// TwinCAT 3 PLC project Untitled1
// ProgramVersion: 3.1.4024.0
// libraries:
//   Tc2_EtherCAT, * (Beckhoff Automation GmbH)
//   Tc2_IoFunctions, * (Beckhoff Automation GmbH)
//   Tc2_Standard, * (Beckhoff Automation GmbH)
//   Tc2_System, * (Beckhoff Automation GmbH)
//   Tc2_Utilities, * (Beckhoff Automation GmbH)
//   Tc3_EventLogger, * (Beckhoff Automation GmbH)
//   Tc3_Module, * (Beckhoff Automation GmbH)
// project tree:
//   / GlobalTextList.TcGTLO, PlcTask.TcTTO, Visualization Manager.TcVMO (not stored), VISU_TASK.TcTTO
//   GVLs/ GVL.TcGVL
//   POUs/EL6910/ FB_SafeDiag_Diagnostic.TcPOU, PH_SafeDiag_DiagHistory_black.TcVIS, PH_SafeDiag_Diagnostic_black.TcVIS, P_Sample.TcPOU, V_SafeDiag_Main.TcVIS
//   POUs/EL6910/Internal/Dedicated/DUTs/ E_SafeLogicState.TcTLEO, ST_EL6910_SafeDiag.TcDUT, ST_SafeDiag_HardwareInfos.TcDUT, ST_SafeDiag_SafetyProjectInfos.TcDUT, ST_SafeDiag_VisualisationInfos.TcDUT
//   POUs/EL6910/Internal/Dedicated/FBs/ FB_HardwareInfos.TcPOU, FB_SafeDiag_Visualisation.TcPOU, FB_SafetyProjectInfos.TcPOU
//   POUs/EL6910/Internal/General/DiagHistory_Events/ FB_DiagHistory_Listener.TcPOU, GVL_DiagHistory_SafetyEvents.TcGVL, ST_DiagHistory_Event.TcDUT
//   POUs/EL6910/Internal/General/EtherCAT/ FB_ReadSlaveBasicInformations.TcPOU, ST_EtherCat_SlaveBasicInfos.TcDUT
//   POUs/EL6910/Internal/General/SafetyEvents/ FB_Listener.TcPOU, FB_SafetyEvents.TcPOU, GVL_SafetyEvents.TcGVL, ST_Event.TcDUT
//   POUs/ MAIN.TcPOU
// real-time tasks:
//   TASK PlcTask: cycle T#10ms, priority 20, ADS port 350
//   TASK VISU_TASK: cycle T#200000us, priority 30, ADS port 351
// I/O:
//   DEVICE Device 1 (EtherCAT), AmsNetId 5.36.73.62.2.1
//     Term 1 (EK1200) [EK1200-5000 EtherCAT Power supply (2A E-Bus)]
//       Term 2 (EL1008) [EL1008 8Ch. Dig. Input 24V, 3ms]
//       Term 3 (EL2008) [EL2008 8Ch. Dig. Output 24V, 0.5A]
//       Term 4 (EL5151) [EL5151 1Ch. Inc. Encoder]
//       Term 5 (EL9110) [EL9110 Power Supplier with LED (24V, Diagnostics)]
//       Term 6 (EL6910) [EL6910, TwinSAFE PLC]
//       Term 7 (EL7037) [EL7037 1Ch. Stepper motor output stage (24V, 1.5A)]
//       Term 8 (EL9512) [EL9512 Power supply terminal 12V]
//       Term 9 (EL3162) [EL3162 2Ch. Ana. Input 0-10V]
//       Term 10 (EL4102) [EL4102 2Ch. Ana. Output  0-10V, 16bit]
//       Term 11 (EK1122) [EK1122 2 port EtherCAT junction]
//         Term 12 (EK1100) [EK1100 EtherCAT Coupler (2A E-Bus)]
//           Term 13 (EL1859) [EL1859 8Ch. Dig. Input 24V, 3ms, 8Ch. Dig. Output 24V, 0.5A]
//           Term 14 (EL1904) [EL1904, 4 Ch. Safety Input 24V, TwinSAFE]
//             modules: Module 1 (FSOES)
//           Term 15 (EL2904) [EL2904, 4 Ch. Safety Output 24V, 0.5A, TwinSAFE]
//             modules: Module 1 (FSOES), Module 2 (DO)
//           Term 16 (EL9110) [EL9110 Power Supplier with LED (24V, Diagnostics)]
//           Term 17 (EL2004) [EL2004 4Ch. Dig. Output 24V, 0.5A]
//           Term 18 (EL9410) [EL9410 E-Bus Power Supplier  (Diagnostics)]
//           Term 19 (EL7201-0010) [EL7201-0010 1Ch. MDP742 Servo motor output stage with OCT (50V, 4A)]
//           Term 27 (EL9011) [EL9011 End Terminal]
//         Term 20 (EK1101) [EK1101 EtherCAT Coupler (2A E-Bus, ID switch)]
//           Term 21 (EL1904) [EL1904, 4 Ch. Safety Input 24V, TwinSAFE]
//             modules: Module 1 (FSOES)
//           Term 22 (EL1252) [EL1252 2Ch. Fast Dig. Input 24V, 1µs, DC Latch]
//           Term 23 (EL1262) [EL1262 2Ch. Dig. Input 24V, 1µs, DC Oversample]
//           Term 24 (EL2252) [EL2252 2Ch. Dig. Output 24V, 0.5A, DC Time Stamp]
//           Term 25 (EL3702) [EL3702 2Ch. Ana. Input +/-10V, DIFF, Oversample]
//           Term 26 (EL4732) [EL4732 2Ch. Ana. Output +/-10V, Oversample]
//           Term 28 (EL9011) [EL9011 End Terminal]
// variable links:
//   Device 1 (EtherCAT) <-> Device 1 (EtherCAT)/Term 1 (EK1200)/Term 11 (EK1122)/Term 12 (EK1100)/Term 15 (EL2904)
//     Term 1 (EK1200)/Term 6 (EL6910)/ConnectionInputs/TwinSafeGroup1.Term 9 (EL2904) - Module 1 (FSOES)_3 TxPDO <-> Module 1 (FSOES)/RxPDO/FSOE
//   Device 1 (EtherCAT) <-> Device 1 (EtherCAT)/Term 1 (EK1200)/Term 6 (EL6910)
//     Term 1 (EK1200)/Term 11 (EK1122)/Term 12 (EK1100)/Term 15 (EL2904)/Module 1 (FSOES)/TxPDO/FSOE <-> ConnectionOutputs/TwinSafeGroup1.Term 9 (EL2904) - Module 1 (FSOES)_3 RxPDO
//   Untitled1/Untitled1 Instance <-> Device 1 (EtherCAT)/Term 1 (EK1200)/Term 6 (EL6910)
//     PlcTask Outputs/GVL.bErrAck <-> StandardOutputs/TwinSafeGroup1.ErrorAcknowledgement_1
//     PlcTask Outputs/GVL.bRun <-> StandardOutputs/TwinSafeGroup1.Run_2

CONFIGURATION Untitled1
    RESOURCE PLC ON TwinCAT3
        TASK PlcTask(INTERVAL := T#10ms, PRIORITY := 20);
        TASK VISU_TASK(INTERVAL := T#200000us, PRIORITY := 30);
        PROGRAM MAIN WITH PlcTask : MAIN;
        PROGRAM VisuElems_Visu_Prg WITH VISU_TASK : VisuElems.Visu_Prg;
    END_RESOURCE
END_CONFIGURATION

// ---- POUs/EL6910/Internal/Dedicated/DUTs/E_SafeLogicState.TcTLEO
{attribute 'qualified_only'}
{attribute 'strict'}
{attribute 'to_string'}
TYPE E_SafeLogicState :
(
	OFFLINE 		:= 0,
	RUN				:= 1,
	STOP			:= 2,
	SAFE			:= 3,
	ERROR           := 4,
	START           := 6,
	PREPARE         := 8,
	RESTORE         := 10,
	PROJECT_CRC_OK  := 11
);
END_TYPE

// ---- POUs/EL6910/Internal/Dedicated/DUTs/ST_EL6910_SafeDiag.TcDUT
TYPE ST_EL6910_SafeDiag :
STRUCT
	stBasicInfo						: ST_EtherCat_SlaveBasicInfos;									// EtherCAT slave basic infos
	stHardwareInfo					: ST_SafeDiag_HardwareInfos;									// Internal module hardware infos
	arrDiagHistory					: ARRAY [1.. GVL_SafetyEvents.MAX_EVENTS] OF ST_Event;			// Event Logger Listener
	stSafetyInfo					: ST_SafeDiag_SafetyProjectInfos;								// Additional Safety informations from Logic Unit
	stVisu							: ST_SafeDiag_VisualisationInfos;								// Internal structure to show gained informations on visualisation
END_STRUCT
END_TYPE

// ---- POUs/EL6910/Internal/Dedicated/DUTs/ST_SafeDiag_HardwareInfos.TcDUT
TYPE ST_SafeDiag_HardwareInfos :
STRUCT
	iVoltageC1				: INT;		// CoE - F985:01	[mV]	
	iVoltageC2				: INT;		// CoE - F984:01	[mV]		
	iTemperatureC1			: INT;		// CoE - F984:02	[Celcius degrees]   
	iTemperatureC2			: INT;		// CoE - F985:02    [Celcius degrees]
END_STRUCT
END_TYPE

// ---- POUs/EL6910/Internal/Dedicated/DUTs/ST_SafeDiag_SafetyProjectInfos.TcDUT
TYPE ST_SafeDiag_SafetyProjectInfos :
STRUCT
	// FSLOGIC status
	wSafeLogicState									: WORD;				// CoE - F100:01
	eSafeLogicState									: E_SafeLogicState; // Reference to CoE F100:01
	wCycleCounter									: WORD;				// CoE - F100:02
	
	// Module internal Safety Task status (CTRL Diag Data)
	uliActualSafetyControlTaskExecution				: ULINT;			// CoE - FEA0:09
	uliMinSafetyControlTaskExecutionTime_Run		: ULINT;  			// CoE - FEA0:0A
	uliMinSafetyControlTaskExecutionTime_NotRun		: ULINT;  			// CoE - FEA0:16
	uliActualSafetyControlTaskExecutionTime_Run		: ULINT;  			// CoE - FEA0:0C
	uliActualSafetyControlTaskExecutionTime_NotRun	: ULINT;  			// CoE - FEA0:15
	
	// Times converted from Distributed Clock Time (DcTime) to TIMSTRUCT
	stActualSafetyControlTaskExecution				: TIMESTRUCT;		// CoE - FEA0:09	(DC Time converted to Timestruct)
	stMinSafetyControlTaskExecutionTime_Run			: TIMESTRUCT;  		// CoE - FEA0:0A    (DC Time converted to Timestruct)
	stMinSafetyControlTaskExecutionTime_NotRun		: TIMESTRUCT;  		// CoE - FEA0:16    (DC Time converted to Timestruct)
	stActualSafetyControlTaskExecutionTime_Run		: TIMESTRUCT;  		// CoE - FEA0:0C    (DC Time converted to Timestruct)
	stActualSafetyControlTaskExecutionTime_NotRun	: TIMESTRUCT;  		// CoE - FEA0:15    (DC Time converted to Timestruct)
END_STRUCT
END_TYPE

// ---- POUs/EL6910/Internal/Dedicated/DUTs/ST_SafeDiag_VisualisationInfos.TcDUT
TYPE ST_SafeDiag_VisualisationInfos :
STRUCT
	// ST_EtherCat_SlaveBasicInfos
	arrBasicInfos						: ARRAY [1..2,1..9] OF STRING(20) := [
												'EtherCat_AmsNetId', 
												'SlaveAdress', 
												'DeviceName', 
												'HardwareVersion', 
												'SoftwareVersion', 
												'VendorId', 
												'ProductCode', 
												'Revision', 
												'SerialNumber'];
	
	
	// ST_SafeDiag_HardwareInfos
	arrHardwareInfos					: ARRAY [1..2, 1..4] OF STRING(20) := [
												'VoltageC1 [mV]', 				 
												'VoltageC2 [mV]', 				 
												'TemperatureC1', 			 
												'TemperatureC2'];

	// ST_SafeDiag_SafetyProjectInfos
	arrSafetyInfos						: ARRAY [1..2, 1..3] OF STRING(20) := [
												'SafeLogicState',
												'SafeLogicState', 				
												'CycleCounter'];
	//Model number
	sModelNumber						:	STRING (20);	

END_STRUCT
END_TYPE

// ---- POUs/EL6910/Internal/General/DiagHistory_Events/ST_DiagHistory_Event.TcDUT
TYPE ST_DiagHistory_Event :
STRUCT
	TimeRaised				: DT;				// Date & time
	eSeverity				: TcEventSeverity;	// Type of message
	EventID					: UDINT;			// Error/warning/message number
	EventText				: STRING(255);		// Error description
END_STRUCT
END_TYPE

// ---- POUs/EL6910/Internal/General/EtherCAT/ST_EtherCat_SlaveBasicInfos.TcDUT
TYPE ST_EtherCat_SlaveBasicInfos :
STRUCT
	// EC Master Infos
	{attribute 'hide'}
	sEtherCat_AmsNetId					: T_AmsNetID;						// EtherCAT master's AmsNetId (usually contain adress IP.2.1)
	{attribute 'hide'}
	arrEcSlaveConfigData				: ARRAY [1..100(* 16#FFFF *)] 	OF  ST_EcSlaveConfigData;
	{attribute 'hide'}
	wSlavesNumber						: WORD	:= 100;						// Slave's number 
	
	
	// EC Slave Infos	
	stSlaveCfgData						: ST_EcSlaveConfigData;
	sHardwareVersion					: STRING;							// CoE	-	16#1009
	sSoftwareVersion					: STRING;							// CoE	-	16#100A
	dwSafetyLogicSerialNo				: DWORD;							// CoE	-	16#F980:02
END_STRUCT
END_TYPE

// ---- POUs/EL6910/Internal/General/SafetyEvents/ST_Event.TcDUT
TYPE ST_Event :
STRUCT
	EventID			: UDINT;
	EventText		: STRING(255);
	Severity		: BYTE;
	TimeRaised		: DT;
END_STRUCT
END_TYPE

// ---- GVLs/GVL.TcGVL
{attribute 'qualified_only'}
VAR_GLOBAL
	bRun		AT%Q* : BOOL;
	bErrAck     AT%Q* : BOOL;
END_VAR

// ---- POUs/EL6910/Internal/General/DiagHistory_Events/GVL_DiagHistory_SafetyEvents.TcGVL
{attribute 'qualified_only'}
VAR_GLOBAL CONSTANT
	MAX_EVENTS				: UINT := 128;	// maximum no. of saved events
	MAX_CURR				: UINT := 10;	// max event occurs at same time
END_VAR

// ---- POUs/EL6910/Internal/General/SafetyEvents/GVL_SafetyEvents.TcGVL
{attribute 'qualified_only'}
VAR_GLOBAL CONSTANT
	MAX_EVENTS				: UINT := 64;	// maximum no. of saved events
	MAX_CURR				: UINT := 10;	// max event occurs at same time
END_VAR

// ---- POUs/MAIN.TcPOU
PROGRAM MAIN
VAR
END_VAR

P_Sample();

END_PROGRAM

// ---- POUs/EL6910/P_Sample.TcPOU
PROGRAM P_Sample
VAR CONSTANT
	sNetID						: T_AmsNetId 	:= '5.36.73.62.2.1'; // EtherCAT Master AMS NetID
	sModule_GUID				: STRING(36)	:= '28111931-0002-0000-5230-FE1A00001100';
END_VAR
VAR
	fbSafeDiag_Diagnostic		: FB_SafeDiag_Diagnostic;
	stSafeDiag					: ST_EL6910_SafeDiag;
	bExecute					: BOOL			:= TRUE;
END_VAR

fbSafeDiag_Diagnostic(
    stSafeDiag := stSafeDiag,
    bExecute := bExecute,
    sEcAmsNetId := sNetID,
    wSlaveAdress := 1005,
    sModule_GUID := sModule_GUID); // FB_SafeDiag_Diagnostic

END_PROGRAM

// ---- POUs/EL6910/FB_SafeDiag_Diagnostic.TcPOU
// ================================================================================================ //
//							Beckhoff Automation Poland                                              //
//									26.03.2021                                                      //
//												                                                    //
//					Function Block to monitor & diagnose safety modules.        					//
//					Function Block works with EL6910, EL2911, EK1960       							//
//												                                                    //
//	FB reads parameters & errors (avaliable also in module's Diag History) via Event Logger         //
// 		Eg. 16#3809 - 	'FB 1 (ESTOP): An DiscTime-Fault (0x0001) was detected in state DELAYOUT, 	//
//						the actual EStopIn-values are 0x0000'                                       //
//                                                                                                  //
//	All data are localised in safety modules           												//
//	                                                                                                //
//	Author: Piotr Szyszka (p.szyszka@beckhoff.pl)                                           		//
//	Requirements: Libraries Tc2_EtherCAT, TC2_Utilities                                    			//
//                                                                                                  //
//  v2.0	|| TC v 3.1.4024.12		||	FB uses Event Listener to get EL6910 Diag Messages			// 
//  v1.0	|| TC v 3.1.4024.7		|| 	First release. Library uses ESI file to find Diag History 	// 
//										Message via JSON lib.                                      	//
// ================================================================================================ //
FUNCTION_BLOCK FB_SafeDiag_Diagnostic
VAR_IN_OUT
	stSafeDiag								: ST_EL6910_SafeDiag;			// Strcture with all informations about EL6910
END_VAR
VAR_INPUT
	bExecute								: BOOL;
	sEcAmsNetId								: T_AmsNetID;			// EtherCAT master's AmsNetId
	wSlaveAdress							: WORD;					// Slave's adress in EtherCAT topology
	sModule_GUID							: STRING(36);			// Event class of module - read from event logger message window (see manual)
END_VAR
VAR_OUTPUT
	bBusy									: BOOL;
	bError									: BOOL;
	udiErrId								: UDINT;
	sError									: STRING;
END_VAR
VAR
	iStep									: INT;
	iLastStep								: INT;
	rtExecute								: R_TRIG;
	iMsg									: INT;
	
	fbReadSlaveBasicInformations			: FB_ReadSlaveBasicInformations;
	fbEL6910_HardwareInfos					: FB_HardwareInfos;
	fbEL6910_SafetyProjectInfos				: FB_SafetyProjectInfos;
	fbSafetyEvents							: FB_SafetyEvents;	
	fbEL6910_Visualisation					: FB_SafeDiag_Visualisation;
END_VAR

rtExecute(CLK:= bExecute, Q=> );
IF rtExecute.Q THEN
	iStep												:= 0;
END_IF

CASE iStep OF
	0:	// Idle
		IF rtExecute.Q THEN
			iLastStep									:= 0;
			bBusy										:= TRUE;
			bError										:= FALSE;
			udiErrId									:= 0;
			sError										:= '';		
			
			fbReadSlaveBasicInformations.bExecute		:= FALSE;
			fbEL6910_HardwareInfos.bExecute				:= FALSE;
			fbEL6910_SafetyProjectInfos.bExecute		:= FALSE;
			
			iStep										:= iStep + 10;
		END_IF
		
	10:	// Read basic informations about EtherCAT slave
		stSafeDiag.stBasicInfo.sEtherCat_AmsNetId			:= sEcAmsNetId;
		fbReadSlaveBasicInformations.bExecute			:= TRUE;
		iStep											:= iStep + 10;
		
	20:	// Wait to gain infos
		fbReadSlaveBasicInformations.bExecute			:= FALSE;
		IF NOT fbReadSlaveBasicInformations.bBusy 	THEN
			IF NOT fbReadSlaveBasicInformations.bError	THEN
				fbEL6910_HardwareInfos.bExecute			:= TRUE;
				iStep									:= iStep + 10;
			ELSE                                		
				udiErrId								:= fbReadSlaveBasicInformations.udiErrId;
				iLastStep								:= iStep;
				iStep									:= 900;
			END_IF
		END_IF
		
	30:	// Read module hardware infos (Voltage, Temp)
		fbEL6910_HardwareInfos.bExecute					:= FALSE;
		IF NOT fbEL6910_HardwareInfos.bBusy THEN
			IF NOT fbEL6910_HardwareInfos.bError THEN
				fbEL6910_SafetyProjectInfos.bExecute	:= TRUE;
				iStep									:= iStep + 10;
			ELSE                                		
				udiErrId								:= fbReadSlaveBasicInformations.udiErrId;
				iLastStep								:= iStep;
				iStep									:= 900;
			END_IF
		END_IF
		
		
	40:	// Read module Safety Project Informations
		fbEL6910_SafetyProjectInfos.bExecute			:= FALSE;
		IF NOT fbEL6910_SafetyProjectInfos.bBusy THEN
			IF NOT fbEL6910_SafetyProjectInfos.bError THEN
				iStep									:= iStep + 10;
			ELSE                               		
				udiErrId								:= fbReadSlaveBasicInformations.udiErrId;
				iLastStep								:= iStep;
				iStep									:= 900;
			END_IF
		END_IF
		
	50:	// Check if DiagHistory - EventLogger has error
		IF NOT fbSafetyEvents.bError THEN
			iStep										:= 100;
		ELSE                               		
			iLastStep									:= iStep;
			iStep										:= 900;
		END_IF
		
	100:	// End procedure
		bBusy											:= FALSE;
		iStep											:= 0;
		
	900:	// Error procedure
		bBusy											:= FALSE;
		bError											:= TRUE;
	ELSE                                        		
		iLastStep										:= iStep;
		iStep											:= 900;
END_CASE


fbReadSlaveBasicInformations(
	stEtherCatSlaveBasicInfos	:= stSafeDiag.stBasicInfo, 
	sEcAmsNetId					:= stSafeDiag.stBasicInfo.sEtherCat_AmsNetId, 
	wSlaveAdress				:= wSlaveAdress);
	
fbEL6910_HardwareInfos(
	stEtherCatSlaveBasicInfos	:= stSafeDiag.stBasicInfo, 
	stHardwareInfo				:= stSafeDiag.stHardwareInfo,
	tAutoRefreshTime			:= T#60S);
	
fbEL6910_SafetyProjectInfos(
	stEtherCatSlaveBasicInfos	:= stSafeDiag.stBasicInfo, 
	stSafetyInfos				:= stSafeDiag.stSafetyInfo,
	tAutoRefreshTime			:= T#5S);
	
fbSafetyEvents(
	sModuleName					:= stSafeDiag.stBasicInfo.stSlaveCfgData.sName, 
	sEventClass					:= sModule_GUID,
	aStEventsData				=> stSafeDiag.arrDiagHistory, 
	bError						=> );

fbEL6910_Visualisation(
	stSafeDiag					:= stSafeDiag, 
	bRefresh					:= , 
	tAutoRefreshTime			:= );

END_FUNCTION_BLOCK

// ---- POUs/EL6910/Internal/General/EtherCAT/FB_ReadSlaveBasicInformations.TcPOU
// ================================================================================================ //
//							Beckhoff Automation Poland                                              //
//									26.03.2021                                                      //
//												                                                    //
//					Function Block to read basic EtherCAT slave infos              					//
//	                                                                                                //
//	Author: Piotr Szyszka (p.szyszka@beckhoff.pl)                                           		//
//	Requirements: Libraries Tc2_EtherCAT 			                                    			//
//                                                                                                  //
//  v1.1	|| TC v 3.1.4024.12		||	Optimalisations												// 
//  v1.0	|| TC v 3.1.4024.7		|| 	First release. 												// 
// ================================================================================================ //
FUNCTION_BLOCK FB_ReadSlaveBasicInformations
VAR_IN_OUT
	stEtherCatSlaveBasicInfos	: ST_EtherCat_SlaveBasicInfos;
END_VAR
VAR_INPUT
	bExecute					: BOOL;
	sEcAmsNetId					: T_AmsNetID;						// EtherCAT master's AmsNetId
	wSlaveAdress				: WORD;								// Certain slave adress in EtherCAT topology to get InfoData
END_VAR
VAR_OUTPUT
	bBusy						: BOOL;
	bError						: BOOL;
	udiErrId					: UDINT;
END_VAR
VAR
	iStep						: INT;
	iLastStep					: INT;
	rtExecute					: R_TRIG;
	i							: INT;
	
	fbEcGetConfSlaves			: FB_EcGetConfSlaves;
	fbEcGetSlaveIdentity		: FB_EcGetSlaveIdentity;
	fbEcCoESdoRead				: FB_EcCoESdoRead;
END_VAR

rtExecute(CLK:= bExecute, Q=> );
IF rtExecute.Q THEN
	iStep												:= 0;
END_IF


CASE iStep OF
	0:	// Idle
		IF rtExecute.Q THEN
			iLastStep									:= 0;
			bBusy										:= TRUE;
			bError										:= FALSE;
			udiErrId									:= 0;
			fbEcGetConfSlaves.bExecute					:= FALSE;
			fbEcGetSlaveIdentity.bExecute				:= FALSE;
			fbEcCoESdoRead.bExecute						:= FALSE;
			                                    		
			stEtherCatSlaveBasicInfos.sEtherCat_AmsNetId:= sEcAmsNetId;
			iStep										:= iStep + 10;
		END_IF
		
	10:	// Get list of configured slaves
		fbEcGetConfSlaves.bExecute						:= TRUE;
		iStep											:= iStep + 10;
			
	20:	// Get slaves identity
		fbEcGetConfSlaves.bExecute						:= FALSE;
		IF NOT fbEcGetConfSlaves.bBusy THEN
			IF NOT fbEcGetConfSlaves.bError THEN
				stEtherCatSlaveBasicInfos.wSlavesNumber	:= fbEcGetConfSlaves.nSlaves;
				iStep									:= iStep + 10;
			ELSE
				udiErrId								:= fbEcGetConfSlaves.nErrorId;
				iLastStep								:= iStep;
				iStep									:= 900;
			END_IF
		END_IF
		
	30:	// Rewrite Slave infos		
		FOR i:=1 TO 	stEtherCatSlaveBasicInfos.wSlavesNumber+1 	DO
			IF wSlaveAdress = stEtherCatSlaveBasicInfos.arrEcSlaveConfigData[i].nAddr THEN
				stEtherCatSlaveBasicInfos.stSlaveCfgData:= stEtherCatSlaveBasicInfos.arrEcSlaveConfigData[i];
				iStep									:= iStep + 10;
				EXIT;
			ELSIF i=stEtherCatSlaveBasicInfos.wSlavesNumber+1 THEN	
				iLastStep								:= iStep;
				iStep									:= 900;	
			END_IF
		END_FOR
		
	40:	// Read module: 	Hardware version
		fbEcCoESdoRead.nIndex 							:= 16#1009;
		fbEcCoESdoRead.nSubIndex 						:= 0;
		fbEcCoESdoRead.pDstBuf 							:= ADR (stEtherCatSlaveBasicInfos.sHardwareVersion);
		fbEcCoESdoRead.cbBufLen 						:= SIZEOF(stEtherCatSlaveBasicInfos.sHardwareVersion);
		fbEcCoESdoRead.bExecute							:= TRUE;
		iStep											:= iStep + 10;
				
	50:	// Read module: 	Software version
		fbEcCoESdoRead.bExecute							:= FALSE;
		IF NOT fbEcCoESdoRead.bBusy THEN
			IF NOT fbEcCoESdoRead.bError THEN
				fbEcCoESdoRead.nIndex 					:= 16#100A;
				fbEcCoESdoRead.nSubIndex 				:= 0;
				fbEcCoESdoRead.pDstBuf 					:= ADR (stEtherCatSlaveBasicInfos.sSoftwareVersion);
				fbEcCoESdoRead.cbBufLen 				:= SIZEOF(stEtherCatSlaveBasicInfos.sSoftwareVersion);
				fbEcCoESdoRead.bExecute					:= TRUE;
				iStep									:= iStep + 10;
			ELSE
				udiErrId								:= fbEcCoESdoRead.nErrId;
				iLastStep								:= iStep;
				iStep									:= 900;
			END_IF
		END_IF
		
	60:	// Read module: 	Safety Logic Serial No
		fbEcCoESdoRead.bExecute							:= FALSE;
		IF NOT fbEcCoESdoRead.bBusy THEN
			IF NOT fbEcCoESdoRead.bError THEN
				fbEcCoESdoRead.nIndex 					:= 16#F980;
				fbEcCoESdoRead.nSubIndex 				:= 2;
				fbEcCoESdoRead.pDstBuf 					:= ADR (stEtherCatSlaveBasicInfos.dwSafetyLogicSerialNo);
				fbEcCoESdoRead.cbBufLen 				:= SIZEOF(stEtherCatSlaveBasicInfos.dwSafetyLogicSerialNo);
				fbEcCoESdoRead.bExecute					:= TRUE;
				iStep									:= iStep + 10;
			ELSE
				udiErrId								:= fbEcCoESdoRead.nErrId;
				iLastStep								:= iStep;
				iStep									:= 900;
			END_IF
		END_IF
		
		
	70:	// // End procedure
		fbEcCoESdoRead.bExecute							:= FALSE;
		IF NOT fbEcCoESdoRead.bBusy THEN
			IF NOT fbEcCoESdoRead.bError THEN
				bBusy									:= FALSE;
				iStep									:= 0;
			ELSE
				udiErrId								:= fbEcCoESdoRead.nErrId;
				iLastStep								:= iStep;
				iStep									:= 900;
			END_IF
		END_IF
		
	900:	// Error procedure
		bBusy											:= FALSE;
		bError											:= TRUE;
	ELSE
		iLastStep										:= iStep;
		iStep											:= 900;
END_CASE


fbEcCoESdoRead(
	sNetId				:= stEtherCatSlaveBasicInfos.sEtherCat_AmsNetId, 
	nSlaveAddr			:= stEtherCatSlaveBasicInfos.stSlaveCfgData.nAddr);

fbEcGetConfSlaves(
	sNetId				:= stEtherCatSlaveBasicInfos.sEtherCat_AmsNetId, 
	pArrEcConfSlaveInfo	:= ADR(stEtherCatSlaveBasicInfos.arrEcSlaveConfigData), 
	cbBufLen			:= SIZEOF(stEtherCatSlaveBasicInfos.arrEcSlaveConfigData) );

END_FUNCTION_BLOCK

// ---- POUs/EL6910/Internal/Dedicated/FBs/FB_HardwareInfos.TcPOU
// ================================================================================================ //
//							Beckhoff Automation Poland                                              //
//									26.03.2021                                                      //
//												                                                    //
//				Function Block to get hardware infos from safety modules							//
//				Function Block works with EL6910, EL2911, EK1960									//
//																									//
//	FB reads parameters & errors (avaliable also in module's Diag History) via Event Logger         //
//                                                                                                  //
//	                                                                                                //
//	Author: Piotr Szyszka (p.szyszka@beckhoff.pl) 													//
//	Requirements: Libraries Tc2_EtherCAT				                                   			//
//                                                                                                  //
//  v1.0	|| TC v 3.1.4024.12		||	First release												// 
// ================================================================================================ //
FUNCTION_BLOCK FB_HardwareInfos
VAR_IN_OUT
	stEtherCatSlaveBasicInfos		: ST_EtherCat_SlaveBasicInfos;
	stHardwareInfo					: ST_SafeDiag_HardwareInfos;
END_VAR
VAR_INPUT
	bExecute						: BOOL;
	tAutoRefreshTime				: TIME		:= T#5S;			// Time to auto-refresh data. Use 0 to disable.
END_VAR
VAR_OUTPUT
	bBusy							: BOOL;
	bError							: BOOL;
	udiErrId						: UDINT;
END_VAR
VAR
	tonRefreshTime					: TON;
	iStep							: INT;
	iLastStep						: INT;
	rtExecute						: R_TRIG;
	fbEcCoESdoRead					: FB_EcCoESdoRead;
END_VAR

IF TIME_TO_DWORD(tAutoRefreshTime) <> 0 THEN
	tonRefreshTime(IN:= NOT tonRefreshTime.Q, PT:= tAutoRefreshTime);
ELSE
	tonRefreshTime(IN:= FALSE);
END_IF

rtExecute(	CLK:= bExecute OR tonRefreshTime.Q, Q=> );
IF rtExecute.Q THEN
	iStep										:= 0;
END_IF


CASE iStep OF
	0:	// Idle
		IF rtExecute.Q THEN
			iLastStep							:= 0;
			bBusy								:= TRUE;
			bError								:= FALSE;
			udiErrId							:= 0;
			fbEcCoESdoRead.bExecute				:= FALSE;
			
			iStep								:= iStep + 10;
		END_IF
		
	10:	// Read module: 	iVoltageC1
		fbEcCoESdoRead.nIndex 					:= 16#F985;
		fbEcCoESdoRead.nSubIndex 				:= 01;
		fbEcCoESdoRead.pDstBuf 					:= ADR (stHardwareInfo.iVoltageC1);
		fbEcCoESdoRead.cbBufLen 				:= SIZEOF(stHardwareInfo.iVoltageC1);
		fbEcCoESdoRead.bExecute					:= TRUE;
		iStep									:= iStep + 10;
		
	20:	// Read module: 	iVoltageC2
		fbEcCoESdoRead.bExecute					:= FALSE;
		IF NOT fbEcCoESdoRead.bBusy THEN
			IF NOT fbEcCoESdoRead.bError THEN
				fbEcCoESdoRead.nIndex 			:= 16#F984;
				fbEcCoESdoRead.nSubIndex 		:= 01;
				fbEcCoESdoRead.pDstBuf 			:= ADR (stHardwareInfo.iVoltageC2);
				fbEcCoESdoRead.cbBufLen 		:= SIZEOF(stHardwareInfo.iVoltageC2);
				fbEcCoESdoRead.bExecute			:= TRUE;
				iStep							:= iStep + 10;
			ELSE
				udiErrId						:= fbEcCoESdoRead.nErrId;
				iLastStep						:= iStep;
				iStep							:= 900;
			END_IF
		END_IF
		
	30:	// Read module: 	iTemperatureC1
		fbEcCoESdoRead.bExecute					:= FALSE;
		IF NOT fbEcCoESdoRead.bBusy THEN
			IF NOT fbEcCoESdoRead.bError THEN
				fbEcCoESdoRead.nIndex 			:= 16#F984;
				fbEcCoESdoRead.nSubIndex 		:= 02;
				fbEcCoESdoRead.pDstBuf 			:= ADR (stHardwareInfo.iTemperatureC1);
				fbEcCoESdoRead.cbBufLen 		:= SIZEOF(stHardwareInfo.iTemperatureC1);
				fbEcCoESdoRead.bExecute			:= TRUE;
				iStep							:= iStep + 10;
			ELSE
				udiErrId						:= fbEcCoESdoRead.nErrId;
				iLastStep						:= iStep;
				iStep							:= 900;
			END_IF
		END_IF
		
	40:	// Read module: 	iTemperatureC2
		fbEcCoESdoRead.bExecute					:= FALSE;
		IF NOT fbEcCoESdoRead.bBusy THEN
			IF NOT fbEcCoESdoRead.bError THEN
				fbEcCoESdoRead.nIndex 			:= 16#F985;
				fbEcCoESdoRead.nSubIndex 		:= 02;
				fbEcCoESdoRead.pDstBuf 			:= ADR (stHardwareInfo.iTemperatureC2);
				fbEcCoESdoRead.cbBufLen 		:= SIZEOF(stHardwareInfo.iTemperatureC2);
				fbEcCoESdoRead.bExecute			:= TRUE;
				iStep							:= iStep + 10;
			ELSE
				udiErrId						:= fbEcCoESdoRead.nErrId;
				iLastStep						:= iStep;
				iStep							:= 900;
			END_IF
		END_IF


	50:	// End procedure
		fbEcCoESdoRead.bExecute					:= FALSE;
		IF NOT fbEcCoESdoRead.bBusy THEN
			IF NOT fbEcCoESdoRead.bError THEN
				bBusy							:= FALSE;
				iStep							:= 0;
			ELSE
				udiErrId						:= fbEcCoESdoRead.nErrId;
				iLastStep						:= iStep;
				iStep							:= 900;
			END_IF
		END_IF

		
		
		
	900:	// Error procedure
		bBusy									:= FALSE;
		bError									:= TRUE;
	ELSE
		iLastStep								:= iStep;
		iStep									:= 900;
END_CASE


fbEcCoESdoRead(
	sNetId			:= stEtherCatSlaveBasicInfos.sEtherCat_AmsNetId, 
	nSlaveAddr		:= stEtherCatSlaveBasicInfos.stSlaveCfgData.nAddr);

END_FUNCTION_BLOCK

// ---- POUs/EL6910/Internal/Dedicated/FBs/FB_SafetyProjectInfos.TcPOU
// ================================================================================================ //
//							Beckhoff Automation Poland                                              //
//									26.03.2021                                                      //
//												                                                    //
//				Function Block to get safety project infos from safety modules						//
//				Function Block works with EL6910, EL2911, EK1960									//
//	                                                                                                	//
//	Author: Piotr Szyszka (p.szyszka@beckhoff.pl) 														//
//	Requirements: Libraries Tc2_EtherCAT				                                   				//
//                                                                                                  	//
//  v1.0	|| TC v 3.1.4024.12		||	First release													//
//	v1.1	|| TC v 3.1.4024.12		||	Fixed adressing for ActualSafetyControlTaskExecutionTime_Run	//
// ====================================================================================================	//
FUNCTION_BLOCK FB_SafetyProjectInfos
VAR_IN_OUT
	stEtherCatSlaveBasicInfos		: ST_EtherCat_SlaveBasicInfos;
	stSafetyInfos					: ST_SafeDiag_SafetyProjectInfos;
END_VAR
VAR_INPUT
	bExecute						: BOOL;
	tAutoRefreshTime				: TIME		:= T#5S;			// Time to auto-refresh data. Use 0 to disable.
END_VAR
VAR_OUTPUT
	bBusy							: BOOL;
	bError							: BOOL;
	udiErrId						: UDINT;
END_VAR
VAR
	tonRefreshTime					: TON;
	iStep							: INT;
	iLastStep						: INT;
	rtExecute						: R_TRIG;
	fbEcCoESdoRead					: FB_EcCoESdoRead;
END_VAR

IF TIME_TO_DWORD(tAutoRefreshTime) <> 0 THEN
	tonRefreshTime(IN:= NOT tonRefreshTime.Q, PT:= tAutoRefreshTime);
ELSE
	tonRefreshTime(IN:= FALSE);
END_IF

rtExecute(CLK:= bExecute OR tonRefreshTime.Q, Q=> );
IF rtExecute.Q THEN
	iStep										:= 0;
END_IF


CASE iStep OF
	0:	// Idle
		IF rtExecute.Q THEN
			iLastStep							:= 0;
			bBusy								:= TRUE;
			bError								:= FALSE;
			udiErrId							:= 0;
			fbEcCoESdoRead.bExecute				:= FALSE;
			
			iStep								:= iStep + 10;
		END_IF
		
		
		
		
	10:	// Read module: 	SafeLogicState
		fbEcCoESdoRead.nIndex 					:= 16#F100;
		fbEcCoESdoRead.nSubIndex 				:= 01;
		fbEcCoESdoRead.pDstBuf 					:= ADR (stSafetyInfos.wSafeLogicState);
		fbEcCoESdoRead.cbBufLen 				:= SIZEOF(stSafetyInfos.wSafeLogicState);
		fbEcCoESdoRead.bExecute					:= TRUE;
		iStep									:= iStep + 10;
		
	20:	// Read module: 	wCycleCounter
		fbEcCoESdoRead.bExecute					:= FALSE;
		IF NOT fbEcCoESdoRead.bBusy THEN
			IF NOT fbEcCoESdoRead.bError THEN
				fbEcCoESdoRead.nIndex 			:= 16#F100;
				fbEcCoESdoRead.nSubIndex 		:= 02;
				fbEcCoESdoRead.pDstBuf 			:= ADR (stSafetyInfos.wCycleCounter);
				fbEcCoESdoRead.cbBufLen 		:= SIZEOF(stSafetyInfos.wCycleCounter);
				fbEcCoESdoRead.bExecute			:= TRUE;
				iStep							:= iStep + 10;
			ELSE
				udiErrId						:= fbEcCoESdoRead.nErrId;
				iLastStep						:= iStep;
				iStep							:= 900;
			END_IF
		END_IF
		
	30:	// E_SafeLogicState
		CASE 	WORD_TO_INT(stSafetyInfos.wSafeLogicState) OF
			E_SafeLogicState.OFFLINE:			stSafetyInfos.eSafeLogicState		:= E_SafeLogicState.OFFLINE;
			E_SafeLogicState.RUN:				stSafetyInfos.eSafeLogicState		:= E_SafeLogicState.RUN;
			E_SafeLogicState.STOP:				stSafetyInfos.eSafeLogicState		:= E_SafeLogicState.STOP;
			E_SafeLogicState.SAFE:				stSafetyInfos.eSafeLogicState		:= E_SafeLogicState.SAFE;
			E_SafeLogicState.ERROR:				stSafetyInfos.eSafeLogicState		:= E_SafeLogicState.ERROR;
			E_SafeLogicState.START:				stSafetyInfos.eSafeLogicState		:= E_SafeLogicState.START;
			E_SafeLogicState.PREPARE:			stSafetyInfos.eSafeLogicState		:= E_SafeLogicState.PREPARE;
			E_SafeLogicState.RESTORE:			stSafetyInfos.eSafeLogicState		:= E_SafeLogicState.RESTORE;
			E_SafeLogicState.PROJECT_CRC_OK:	stSafetyInfos.eSafeLogicState		:= E_SafeLogicState.PROJECT_CRC_OK;
		END_CASE
		iStep							:= iStep + 10;
		
	40:	// Read module: 	wActualSafetyControlTaskExecution
		fbEcCoESdoRead.nIndex 					:= 16#FEA0;
		fbEcCoESdoRead.nSubIndex 				:= 09;
		fbEcCoESdoRead.pDstBuf 					:= ADR (stSafetyInfos.uliActualSafetyControlTaskExecution);
		fbEcCoESdoRead.cbBufLen 				:= SIZEOF(stSafetyInfos.uliActualSafetyControlTaskExecution);
		fbEcCoESdoRead.bExecute					:= TRUE;
		iStep									:= iStep + 10;
		
	50:	// Read module: 	wMinSafetyControlTaskExecutionTime_Run
		fbEcCoESdoRead.bExecute					:= FALSE;
		IF NOT fbEcCoESdoRead.bBusy THEN
			IF NOT fbEcCoESdoRead.bError THEN
				fbEcCoESdoRead.nIndex 			:= 16#FEA0;
				fbEcCoESdoRead.nSubIndex 		:= 16#0A;
				fbEcCoESdoRead.pDstBuf 			:= ADR (stSafetyInfos.uliMinSafetyControlTaskExecutionTime_Run);
				fbEcCoESdoRead.cbBufLen 		:= SIZEOF(stSafetyInfos.uliMinSafetyControlTaskExecutionTime_Run);
				fbEcCoESdoRead.bExecute			:= TRUE;
				iStep							:= iStep + 10;
			ELSE
				udiErrId						:= fbEcCoESdoRead.nErrId;
				iLastStep						:= iStep;
				iStep							:= 900;
			END_IF
		END_IF
		
	60:	// Read module: 	wMinSafetyControlTaskExecutionTime_NotRun
		fbEcCoESdoRead.bExecute					:= FALSE;
		IF NOT fbEcCoESdoRead.bBusy THEN
			IF NOT fbEcCoESdoRead.bError THEN
				fbEcCoESdoRead.nIndex 			:= 16#FEA0;
				fbEcCoESdoRead.nSubIndex 		:= 16#16;
				fbEcCoESdoRead.pDstBuf 			:= ADR (stSafetyInfos.uliMinSafetyControlTaskExecutionTime_NotRun);
				fbEcCoESdoRead.cbBufLen 		:= SIZEOF(stSafetyInfos.uliMinSafetyControlTaskExecutionTime_NotRun);
				fbEcCoESdoRead.bExecute			:= TRUE;
				iStep							:= iStep + 10;
			ELSE
				udiErrId						:= fbEcCoESdoRead.nErrId;
				iLastStep						:= iStep;
				iStep							:= 900;
			END_IF
		END_IF
		
	70:	// Read module: 	wActualSafetyControlTaskExecutionTime_Run
		fbEcCoESdoRead.bExecute					:= FALSE;
		IF NOT fbEcCoESdoRead.bBusy THEN
			IF NOT fbEcCoESdoRead.bError THEN
				fbEcCoESdoRead.nIndex 			:= 16#FEA0;
				fbEcCoESdoRead.nSubIndex 		:= 16#0C;
				fbEcCoESdoRead.pDstBuf 			:= ADR (stSafetyInfos.uliActualSafetyControlTaskExecutionTime_Run);
				fbEcCoESdoRead.cbBufLen 		:= SIZEOF(stSafetyInfos.uliActualSafetyControlTaskExecutionTime_Run);
				fbEcCoESdoRead.bExecute			:= TRUE;
				iStep							:= iStep + 10;
			ELSE
				udiErrId						:= fbEcCoESdoRead.nErrId;
				iLastStep						:= iStep;
				iStep							:= 900;
			END_IF
		END_IF
		
	80:	// Read module: 	wActualSafetyControlTaskExecutionTime_NotRun
		fbEcCoESdoRead.bExecute					:= FALSE;
		IF NOT fbEcCoESdoRead.bBusy THEN
			IF NOT fbEcCoESdoRead.bError THEN
				fbEcCoESdoRead.nIndex 			:= 16#FEA0;
				fbEcCoESdoRead.nSubIndex 		:= 16#15;
				fbEcCoESdoRead.pDstBuf 			:= ADR (stSafetyInfos.uliActualSafetyControlTaskExecutionTime_NotRun);
				fbEcCoESdoRead.cbBufLen 		:= SIZEOF(stSafetyInfos.uliActualSafetyControlTaskExecutionTime_NotRun);
				fbEcCoESdoRead.bExecute			:= TRUE;
				iStep							:= iStep + 10;
			ELSE
				udiErrId						:= fbEcCoESdoRead.nErrId;
				iLastStep						:= iStep;
				iStep							:= 900;
			END_IF
		END_IF
		
	90:	// Wait for gain infos
		fbEcCoESdoRead.bExecute					:= FALSE;
		IF NOT fbEcCoESdoRead.bBusy THEN
			IF NOT fbEcCoESdoRead.bError THEN
				iStep							:= iStep + 10;
			ELSE
				udiErrId						:= fbEcCoESdoRead.nErrId;
				iLastStep						:= iStep;
				iStep							:= 900;
			END_IF
		END_IF
		
	100:	// DC conversions
		stSafetyInfos.stActualSafetyControlTaskExecution				:=	
			DCTIME64_TO_SYSTEMTIME(stSafetyInfos.uliActualSafetyControlTaskExecution);
		
		stSafetyInfos.stMinSafetyControlTaskExecutionTime_Run			:=
			DCTIME64_TO_SYSTEMTIME(stSafetyInfos.uliMinSafetyControlTaskExecutionTime_Run);
		
		
		stSafetyInfos.stMinSafetyControlTaskExecutionTime_NotRun		:=
			DCTIME64_TO_SYSTEMTIME(stSafetyInfos.uliMinSafetyControlTaskExecutionTime_NotRun);
		
		
		stSafetyInfos.stActualSafetyControlTaskExecutionTime_Run		:=
			DCTIME64_TO_SYSTEMTIME(stSafetyInfos.uliActualSafetyControlTaskExecutionTime_Run);
		
		
		stSafetyInfos.stActualSafetyControlTaskExecutionTime_NotRun     :=
			DCTIME64_TO_SYSTEMTIME(stSafetyInfos.uliActualSafetyControlTaskExecutionTime_NotRun);
		
			
			
		bBusy									:= FALSE;
		iStep									:= 0;
		
		
	900:	// Error procedure
		bBusy									:= FALSE;
		bError									:= TRUE;
	ELSE
		iLastStep								:= iStep;
		iStep									:= 900;
END_CASE


fbEcCoESdoRead(
	sNetId			:= stEtherCatSlaveBasicInfos.sEtherCat_AmsNetId, 
	nSlaveAddr		:= stEtherCatSlaveBasicInfos.stSlaveCfgData.nAddr);

END_FUNCTION_BLOCK

// ---- POUs/EL6910/Internal/General/SafetyEvents/FB_SafetyEvents.TcPOU
FUNCTION_BLOCK FB_SafetyEvents
VAR_INPUT
	sModuleName			: STRING;		// module name, for example: EL6910 - 'Term 6 (EL6910)'
	sEventClass			: STRING(36);	// event class of module, for example: EL6910 - '28111931-0002-0000-5230-FE1A00001100'
END_VAR
VAR_OUTPUT
	aStEventsData		: ARRAY [1..GVL_SafetyEvents.MAX_EVENTS] OF ST_Event;	// output structure with saved events
	bError				: BOOL;			// error flag
END_VAR
VAR
	hr					: HRESULT;
	hrLastError			: HRESULT;

	sLastModuleName		: STRING;	
    sLastEventClass		: STRING(36);
	
	ipMessageConfig		: ITcEventFilterConfig;	// filter interface
	guidEventClass		: GUID;			// GUID of device
	fbListener			: FB_Listener;	// extended listener fb
END_VAR

IF sModuleName <> sLastModuleName OR sEventClass <> sLastEventClass THEN
	// Save last values
	sLastModuleName := sModuleName;
	sLastEventClass := sEventClass;
	
	// Clear output
	fbListener.ClearOutput();
	
	// Remove listener to module event class
	IF ipMessageConfig <> 0 THEN
		fbListener.Unsubscribe();
	END_IF
	
	// Convert event class to GUID
	guidEventClass := STRING_TO_GUID(sEventClass);
	
	// Pass event source filter
	fbListener.sSourceFilter := sModuleName;
	
	// If GUID is not empty, and so on...
	IF GUID_TO_STRING(guidEventClass) <> GUID_TO_STRING(EMPTY_EVENT_CLASS) AND sModuleName <> '' THEN	
		// Reset error flag
		bError := FALSE;
		
		// Add listener to module event class
		fbListener.Subscribe(ADR(ipMessageConfig), 0);
		IF (ipMessageConfig <> 0) THEN
			ipMessageConfig.AddEventClass(guidEventClass, TcEventSeverity.Verbose);
		END_IF
	ELSE
		// Set error flag
		bError := TRUE;
	END_IF
END_IF

// Listener cyclic execute
fbListener.Execute();
	
// Pass outputs from listener
aStEventsData			:= fbListener.aStSavedEvents;

END_FUNCTION_BLOCK

// ---- POUs/EL6910/Internal/General/SafetyEvents/FB_Listener.TcPOU
FUNCTION_BLOCK FB_Listener EXTENDS FB_ListenerBase2
VAR_INPUT
	sSourceFilter			: STRING;	// filter events by this source
END_VAR

VAR_OUTPUT
	aStSavedEvents			: ARRAY [1..GVL_SafetyEvents.MAX_EVENTS] OF ST_Event;	// output array
END_VAR

VAR
	nCntMessagesSent		: UINT;		// messages sent counter
	nCntMessagesNow			: UINT;		// messages sent at once counter
	nCntMessagesSaved		: UINT;		// messages saved in output array counter
	
	nCntRequestReturn		: UINT;		// internal counter, used to delay output queue, and get event text before
	
	nIdx					: UINT;		// index, used in for loops
	
	bReqText				: ARRAY [1..GVL_SafetyEvents.MAX_CURR] OF BOOL;	// request event text flag
	
	aStCachedEvents			: ARRAY [1..GVL_SafetyEvents.MAX_CURR] OF ST_Event;	// cached event structure
	
	SystemTime				: T_FILETIME;						// system time structure
	fbGetSystemTime			: GETSYSTEMTIME;					// get system time fb
	fbRequestEventText		: ARRAY [1..GVL_SafetyEvents.MAX_CURR] OF FB_RequestEventText;	// request event text fb
END_VAR

METHOD ClearOutput : HRESULT
VAR_INPUT
END_VAR
MEMSET(ADR(aStSavedEvents), 16#00, SIZEOF(aStSavedEvents));
END_METHOD

METHOD Execute : HRESULT
// Retrieve events
Execute := SUPER^.Execute();

// Reset retrieved text counter
nCntRequestReturn := 0;

// Retrieve the text of queued messages
FOR nIdx := 1 TO nCntMessagesNow DO
	// If requested, and error
	IF 	bReqText[nIdx] AND fbRequestEventText[nIdx].bError THEN
		// Reset request flag
		bReqText[nIdx] := FALSE;
		// Show error message
		aStCachedEvents[nIdx].EventText := 'Error retrieve event text';
		nCntRequestReturn := nCntRequestReturn + 1;
	// If requested and retrieved
	ELSIF bReqText[nIdx] AND NOT fbRequestEventText[nIdx].bBusy THEN
		// Get retrieved text
		fbRequestEventText[nIdx].GetString(aStCachedEvents[nIdx].EventText, SIZEOF(aStCachedEvents[nIdx].EventText));
		// Reset request flag
		bReqText[nIdx] := FALSE;
		// Increase retrieved text counter
		nCntRequestReturn := nCntRequestReturn + 1;
	END_IF
END_FOR

// If catched events are present, and all requests are retrevied ...
IF nCntMessagesSent > nCntMessagesSaved AND nCntRequestReturn = nCntMessagesNow THEN
	// Reset catched events number
	nCntMessagesSaved := nCntMessagesSent;
	// Move output array
	MEMMOVE(ADR(aStSavedEvents[nCntMessagesNow + 1]), ADR(aStSavedEvents[1]), SIZEOF(aStSavedEvents[1]) * (GVL_SafetyEvents.MAX_CURR - nCntMessagesNow));
	// Move catched events to output array
	FOR nIdx := 1 TO nCntMessagesNow DO
		aStSavedEvents[nIdx] := aStCachedEvents[nIdx];
	END_FOR
	// Reset current catched events counter
	nCntMessagesNow := 0;
END_IF
END_METHOD

METHOD OnMessageSent : HRESULT

VAR_INPUT
	fbEvent : REFERENCE TO FB_TcEvent;
END_VAR
// If source is different that desired module, skip this event
IF fbEvent.ipSourceInfo.sName = sSourceFilter THEN
	// If possible, count handled events
	IF (nCntMessagesSent + 1) < 65535 THEN
		nCntMessagesSent	:= nCntMessagesSent + 1;
	// If counter overflow, reset counters and continue work ...
	ELSE
		nCntMessagesSent	:= 1;
		nCntMessagesSaved	:= 0;
	END_IF
	
	// If messages at once are less than max...
	IF nCntMessagesNow + 1 <= GVL_SafetyEvents.MAX_CURR THEN
		// Increase messages at once counter (if no delay between events, this method will be called more than once, so we use iterator to handle more events at once)
		nCntMessagesNow	:= nCntMessagesNow + 1;
		
		// Request event text
		fbRequestEventText[nCntMessagesNow].Request(
			eventClass	:= fbEvent.EventClass,
			nEventId	:= fbEvent.nEventId,
			nLangId		:= 1033,
			ipArgs		:= fbEvent.ipArguments
		);
		
		// Set request flag
		bReqText[nCntMessagesNow] := TRUE;
		
		// Save event data
		aStCachedEvents[nCntMessagesNow].EventID	:= fbEvent.nEventId;
		aStCachedEvents[nCntMessagesNow].Severity	:= TO_BYTE(fbEvent.eSeverity);
		
		// Get current system time
		fbGetSystemTime(
			timeLoDW => SystemTime.dwLowDateTime,
			timeHiDW => SystemTime.dwHighDateTime );
		
		// Save current system time, as event raised time
		aStCachedEvents[nCntMessagesNow].TimeRaised	:= FILETIME_TO_DT(SystemTime); // Convert time to DateTime format
	
		// Set output
		OnMessageSent	:= S_OK; // in order to receive more callbacks (Set <> S_OK in order to cancel the callbacks for this program cycle.)
	ELSE
		OnMessageSent	:= E_FAIL;
	END_IF
END_IF
END_METHOD

END_FUNCTION_BLOCK

// ---- POUs/EL6910/Internal/Dedicated/FBs/FB_SafeDiag_Visualisation.TcPOU
// ================================================================================================ //
//							Beckhoff Automation Poland                                              //
//									26.03.2021                                                      //
//												                                                    //
//				Function Block to visualise all gained safety module diag data.						//
//				Function Block works with EL6910, EL2911, EK1960									//
//                                                                                                  //
//	                                                                                                //
//	Author: Piotr Szyszka (p.szyszka@beckhoff.pl) 													//
//	Requirements: Libraries Tc2_EtherCAT				                                   			//
//                                                                                                  //
//  v1.0	|| TC v 3.1.4024.12		||	First release												// 
// ================================================================================================ //
FUNCTION_BLOCK FB_SafeDiag_Visualisation
VAR_IN_OUT
	stSafeDiag						: ST_EL6910_SafeDiag;			// Strcture with all informations about EL6910
END_VAR
VAR_INPUT
	bRefresh						: BOOL;
	tAutoRefreshTime				: TIME		:= T#5S;	// Time to auto-refresh data. Use 0 to disable.
END_VAR
VAR_OUTPUT
END_VAR
VAR
	wAddr							:WORD;
	tonRefreshTime					: TON;
	bFillBasicInfo					: BOOL	:= TRUE;
	i								: INT;
END_VAR

tonRefreshTime(IN:= NOT tonRefreshTime.Q, PT:= tAutoRefreshTime, Q=> , ET=> );

IF tonRefreshTime.Q OR bRefresh THEN
	// ST_EtherCat_SlaveBasicInfos
	IF bFillBasicInfo OR (wAddr<>stSafeDiag.stBasicInfo.stSlaveCfgData.nAddr) THEN
		stSafeDiag.stVisu.arrBasicInfos[2,1]			:= stSafeDiag.stBasicInfo.sEtherCat_AmsNetId;
		stSafeDiag.stVisu.arrBasicInfos[2,2]			:= WORD_TO_STRING(stSafeDiag.stBasicInfo.stSlaveCfgData.nAddr);
		stSafeDiag.stVisu.arrBasicInfos[2,3]			:= stSafeDiag.stBasicInfo.stSlaveCfgData.sName;
		stSafeDiag.stVisu.arrBasicInfos[2,4]			:= stSafeDiag.stBasicInfo.sHardwareVersion;
		stSafeDiag.stVisu.arrBasicInfos[2,5]			:= stSafeDiag.stBasicInfo.sSoftwareVersion;
		stSafeDiag.stVisu.arrBasicInfos[2,6]			:= DWORD_TO_STRING(stSafeDiag.stBasicInfo.stSlaveCfgData.stSlaveIdentity.vendorId); 
		stSafeDiag.stVisu.arrBasicInfos[2,7]			:= CONCAT('0x', 	DWORD_TO_HEXSTR(	in	:= stSafeDiag.stBasicInfo.stSlaveCfgData.stSlaveIdentity.productCode, iPrecision :=  8, 	bLoCase := FALSE));
		stSafeDiag.stVisu.arrBasicInfos[2,8]			:= CONCAT('0x', 	DWORD_TO_HEXSTR(	in	:= stSafeDiag.stBasicInfo.stSlaveCfgData.stSlaveIdentity.revisionNo, 	iPrecision :=  8, 	bLoCase := FALSE)); 
		stSafeDiag.stVisu.arrBasicInfos[2,9]			:= CONCAT('0x', 	DWORD_TO_HEXSTR(	in	:= stSafeDiag.stBasicInfo.dwSafetyLogicSerialNo, 	iPrecision :=  8, 	bLoCase := FALSE));
		stSafeDiag.stVisu.sModelNumber				:= MID(stSafeDiag.stBasicInfo.stSlaveCfgData.sName,6,(FIND(stSafeDiag.stBasicInfo.stSlaveCfgData.sName,'(')+1));
		wAddr										:=stSafeDiag.stBasicInfo.stSlaveCfgData.nAddr;
		FOR i := 1 TO 9 DO
			IF stSafeDiag.stVisu.arrBasicInfos[2, i] = '' THEN
				EXIT;
			ELSE
				IF i = 9 THEN
					bFillBasicInfo					:= FALSE;
				END_IF
			END_IF
		END_FOR
	END_IF
	
	
	// ST_SafeDiag_HardwareInfos
		stSafeDiag.stVisu.arrHardwareInfos[2,1]		:= INT_TO_STRING(stSafeDiag.stHardwareInfo.iVoltageC1);
		stSafeDiag.stVisu.arrHardwareInfos[2,2]       := INT_TO_STRING(stSafeDiag.stHardwareInfo.iVoltageC2);
		stSafeDiag.stVisu.arrHardwareInfos[2,3]       := INT_TO_STRING(stSafeDiag.stHardwareInfo.iTemperatureC1);
		stSafeDiag.stVisu.arrHardwareInfos[2,4]       := INT_TO_STRING(stSafeDiag.stHardwareInfo.iTemperatureC2);
	
	// ST_SafeDiag_SafetyProjectInfos
		stSafeDiag.stVisu.arrSafetyInfos[2,1]			:= WORD_TO_STRING(stSafeDiag.stSafetyInfo.wSafeLogicState);
		stSafeDiag.stVisu.arrSafetyInfos[2,2]			:= TO_STRING(stSafeDiag.stSafetyInfo.eSafeLogicState);
		stSafeDiag.stVisu.arrSafetyInfos[2,3]			:= WORD_TO_STRING(stSafeDiag.stSafetyInfo.wCycleCounter);
		
END_IF

END_FUNCTION_BLOCK

// ---- POUs/EL6910/Internal/General/DiagHistory_Events/FB_DiagHistory_Listener.TcPOU
// ================================================================================================ //
//							Beckhoff Automation Poland                                              //
//									26.03.2021                                                      //
//												                                                    //
//				Function Block to get certain Event Logger messages from EterCAT slave				//
//												                                                    //
//	FB reads parameters & errors (avaliable also in module's Diag History) via Event Logger         //
// 		Eg. 16#3809 - 	'FB 1 (ESTOP): An DiscTime-Fault (0x0001) was detected in state DELAYOUT, 	//
//						the actual EStopIn-values are 0x0000'                                       //
//                                                                                                  //
//	                                                                                                //
//	Author: Piotr Szyszka (p.szyszka@beckhoff.pl) & Patryk Supel (p.supel@beckhoff.pl)				//
//	Requirements: Libraries Tc3_EventLogger				                                   			//
//                                                                                                  //
//  v1.0	|| TC v 3.1.4024.12		||	First release												// 
// ================================================================================================ //
FUNCTION_BLOCK FB_DiagHistory_Listener EXTENDS FB_ListenerBase2
VAR_INPUT
	sSourceFilter			: STRING;	// filter events by this source
END_VAR

VAR_OUTPUT
	aStSavedEvents			: ARRAY [1..GVL_DiagHistory_SafetyEvents.MAX_EVENTS] OF ST_DiagHistory_Event;	// output array
END_VAR

VAR
	nCntMessagesSent		: UINT;		// messages sent counter
	nCntMessagesNow			: UINT;		// messages sent at once counter
	nCntMessagesSaved		: UINT;		// messages saved in output array counter
	
	nCntRequestReturn		: UINT;		// internal counter, used to delay output queue, and get event text before
	
	nIdx					: UINT;		// index, used in for loops
	
	bReqText				: ARRAY [1..GVL_DiagHistory_SafetyEvents.MAX_CURR] OF BOOL;	// request event text flag
	
	aStCachedEvents			: ARRAY [1..GVL_DiagHistory_SafetyEvents.MAX_CURR] OF ST_DiagHistory_Event;	// cached event structure
	
	SystemTime				: T_FILETIME;						// system time structure
	fbGetSystemTime			: GETSYSTEMTIME;					// get system time fb
	fbRequestEventText		: ARRAY [1..GVL_DiagHistory_SafetyEvents.MAX_CURR] OF FB_RequestEventText;	// request event text fb
END_VAR

METHOD ClearOutput : HRESULT
VAR_INPUT
END_VAR
MEMSET(ADR(aStSavedEvents), 16#00, SIZEOF(aStSavedEvents));
END_METHOD

METHOD Execute : HRESULT
// Retrieve events
Execute := SUPER^.Execute();

// Reset retrieved text counter
nCntRequestReturn := 0;

// Retrieve the text of queued messages
FOR nIdx := 1 TO nCntMessagesNow DO
	// If requested, and error
	IF 	bReqText[nIdx] AND fbRequestEventText[nIdx].bError THEN
		// Reset request flag
		bReqText[nIdx] := FALSE;
		// Show error message
		aStCachedEvents[nIdx].EventText := 'Error retrieve event text';
		nCntRequestReturn := nCntRequestReturn + 1;
	// If requested and retrieved
	ELSIF bReqText[nIdx] AND NOT fbRequestEventText[nIdx].bBusy THEN
		// Get retrieved text
		fbRequestEventText[nIdx].GetString(aStCachedEvents[nIdx].EventText, SIZEOF(aStCachedEvents[nIdx].EventText));
		// Reset request flag
		bReqText[nIdx] := FALSE;
		// Increase retrieved text counter
		nCntRequestReturn := nCntRequestReturn + 1;
	END_IF
END_FOR

// If catched events are present, and all requests are retrevied ...
IF nCntMessagesSent > nCntMessagesSaved AND nCntRequestReturn = nCntMessagesNow THEN
	// Reset catched events number
	nCntMessagesSaved := nCntMessagesSent;
	// Move output array
	MEMMOVE(ADR(aStSavedEvents[nCntMessagesNow + 1]), ADR(aStSavedEvents[1]), SIZEOF(aStSavedEvents[1]) * (GVL_DiagHistory_SafetyEvents.MAX_CURR - nCntMessagesNow));
	// Move catched events to output array
	FOR nIdx := 1 TO nCntMessagesNow DO
		aStSavedEvents[nIdx] := aStCachedEvents[nIdx];
	END_FOR
	// Reset current catched events counter
	nCntMessagesNow := 0;
END_IF
END_METHOD

METHOD OnMessageSent : HRESULT

VAR_INPUT
	fbEvent : REFERENCE TO FB_TcEvent;
END_VAR
// If source is different that desired module, skip this event
IF fbEvent.ipSourceInfo.sName = sSourceFilter THEN
	// If possible, count handled events
	IF (nCntMessagesSent + 1) < 65535 THEN
		nCntMessagesSent	:= nCntMessagesSent + 1;
	// If counter overflow, reset counters and continue work ...
	ELSE
		nCntMessagesSent	:= 1;
		nCntMessagesSaved	:= 0;
	END_IF
	
	// If messages at once are less than max...
	IF nCntMessagesNow + 1 <= GVL_DiagHistory_SafetyEvents.MAX_CURR THEN
		// Increase messages at once counter (if no delay between events, this method will be called more than once, so we use iterator to handle more events at once)
		nCntMessagesNow	:= nCntMessagesNow + 1;
		
		// Request event text
		fbRequestEventText[nCntMessagesNow].Request(
			eventClass	:= fbEvent.EventClass,
			nEventId	:= fbEvent.nEventId,
			nLangId		:= 1033,
			ipArgs		:= fbEvent.ipArguments
		);
		
		// Set request flag
		bReqText[nCntMessagesNow] := TRUE;
		
		// Save event data
		aStCachedEvents[nCntMessagesNow].EventID	:= fbEvent.nEventId;
		aStCachedEvents[nCntMessagesNow].eSeverity	:= fbEvent.eSeverity;
		
		// Get current system time
		fbGetSystemTime(
			timeLoDW => SystemTime.dwLowDateTime,
			timeHiDW => SystemTime.dwHighDateTime );
		
		// Save current system time, as event raised time
		aStCachedEvents[nCntMessagesNow].TimeRaised	:= FILETIME_TO_DT(SystemTime); // Convert time to DateTime format
	
		// Set output
		OnMessageSent	:= S_OK; // in order to receive more callbacks (Set <> S_OK in order to cancel the callbacks for this program cycle.)
	ELSE
		OnMessageSent	:= E_FAIL;
	END_IF
END_IF
END_METHOD

END_FUNCTION_BLOCK

// ---- GlobalTextList.TcGTLO
TEXTLIST GlobalTextList
  902 = '%s'
  506 = "'Event Text'"
  427 = "'EventID'"
  364 = "'Severity'"
  885 = "'Time Raised'"
  1311 = 'Basic Info'
  1371 = 'BECKHOFF'
  1022 = 'bExec EL2911_Diag'
  139 = 'DiagHistory error list'
  886 = 'EL6910'
  694 = 'Error Code'
  695 = 'Error Description'
  884 = 'Event Text'
  287 = 'EventID'
  542 = 'EventText'
  440 = 'Execute'
  1329 = 'Hardware Info'
  1526 = 'Safety Info'
  693 = 'Severity'
  692 = 'Time Raised'
  393 = 'TimeRaised'
END_TEXTLIST

// ---- POUs/EL6910/PH_SafeDiag_DiagHistory_black.TcVIS
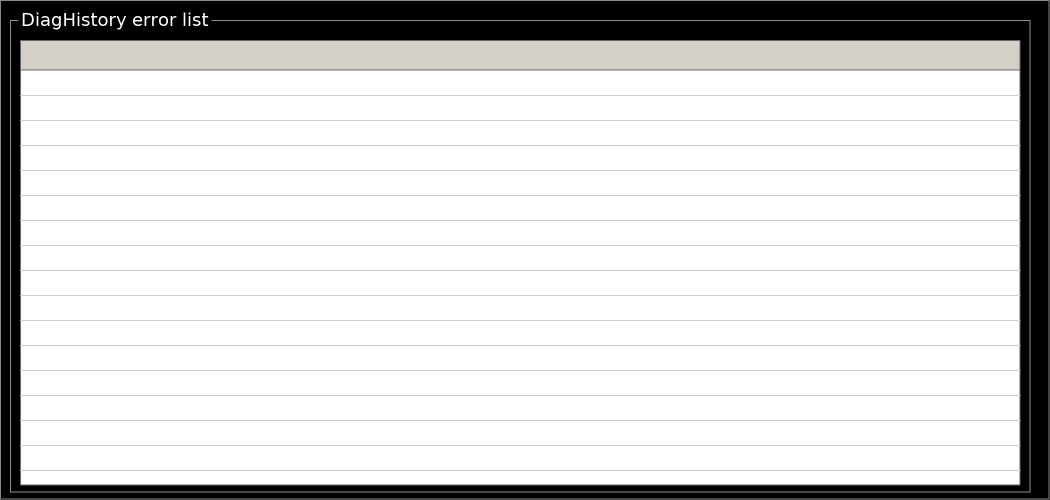
VISUALIZATION PH_SafeDiag_DiagHistory_black  // 1050x500
    GroupBox (10,12 1020x480), "DiagHistory error list"
        Table (10,28 1000x445), data array: P_Sample.stSafeDiag.arrDiagHistory
            p3854506369: P_Sample.stSafeDiag.arrDiagHistory[INDEX].EventID
            p1892666644: P_Sample.stSafeDiag.arrDiagHistory[INDEX].EventText
            p338671338: P_Sample.stSafeDiag.arrDiagHistory[INDEX].Severity
            p2170511999: P_Sample.stSafeDiag.arrDiagHistory[INDEX].TimeRaised
            p3723444502: MAINSafety.stEL6910.stVisu
END_VISUALIZATION

// ---- POUs/EL6910/PH_SafeDiag_Diagnostic_black.TcVIS
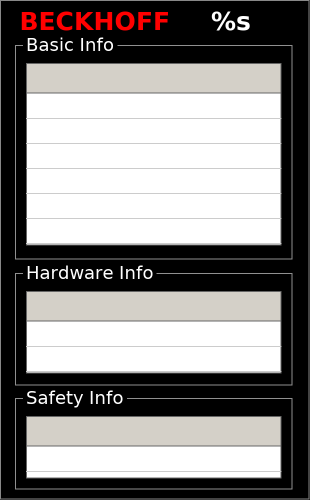
VISUALIZATION PH_SafeDiag_Diagnostic_black  // 310x500
VAR_IN_OUT
	stVisu						: ST_SafeDiag_VisualisationInfos;		
	stSafeDiag					: ST_EL6910_SafeDiag;
END_VAR
    Textfield (10,1 170x40), "BECKHOFF"
    Textfield (171,1 120x40), "%s", text variable: stVisu.sModelNumber
    GroupBox (15,37 277x222), "Basic Info"
        Table (11,26 255x182), data array: stVisu.arrBasicInfos
            p3854506369: stVisu.arrBasicInfos[1,INDEX]
            p1892666644: stVisu.arrBasicInfos[2,INDEX]
    GroupBox (15,265 277x120), "Hardware Info"
        Table (11,26 255x82), data array: stVisu.arrHardwareInfos
            p3854506369: stVisu.arrHardwareInfos[1,INDEX]
            p1892666644: stVisu.arrHardwareInfos[2,INDEX]
    GroupBox (15,390 277x99), "Safety Info"
        Table (11,26 255x62), data array: stVisu.arrSafetyInfos
            p3854506369: stVisu.arrSafetyInfos[1,INDEX]
            p1892666644: stVisu.arrSafetyInfos[2,INDEX]
END_VISUALIZATION

// ---- POUs/EL6910/V_SafeDiag_Main.TcVIS
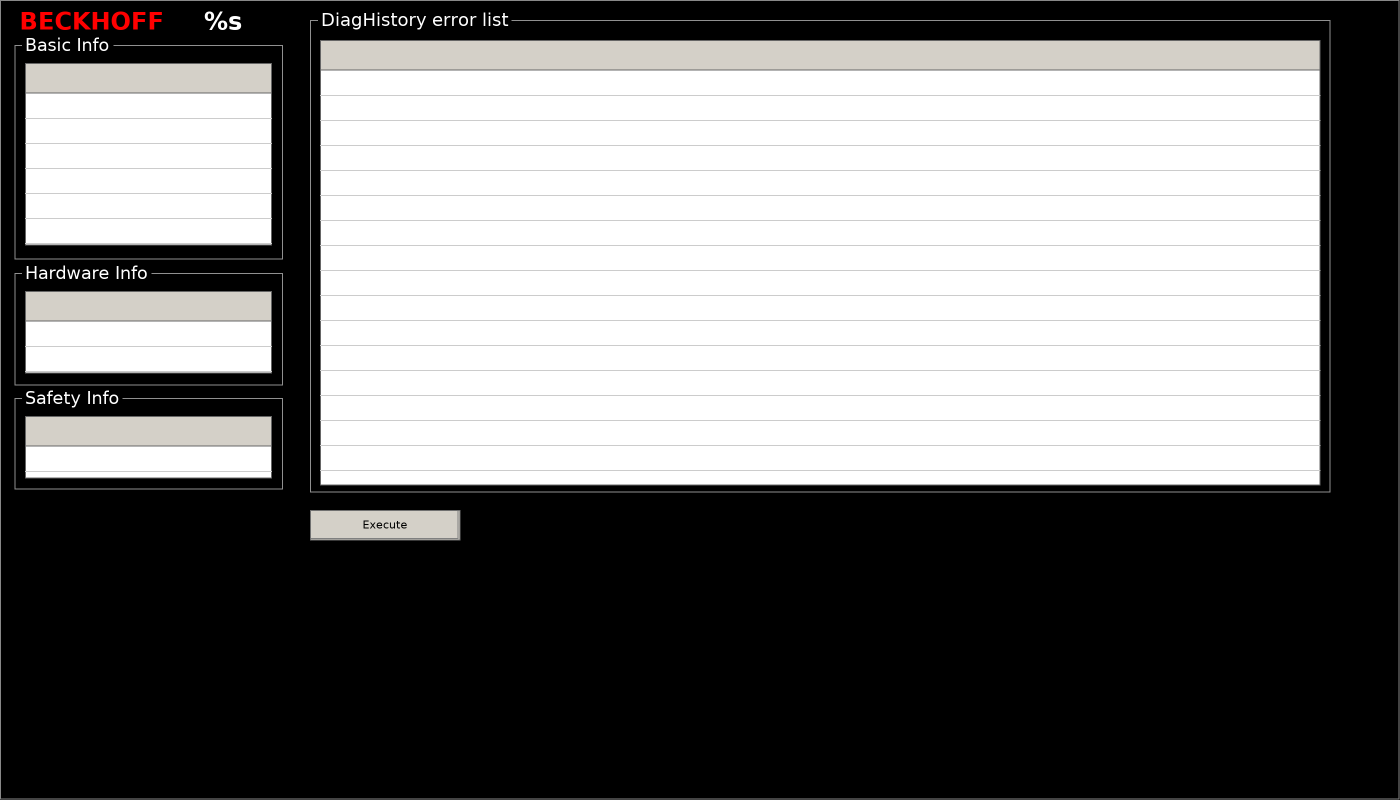
VISUALIZATION V_SafeDiag_Main  // 1400x800
    Button (310,510 150x30), "Execute"
        tap P_Sample.bExecute
    Frame (0,0 300x500)
        shows PH_SafeDiag_Diagnostic_black(stVisu := P_Sample.stSafeDiag.stVisu, stSafeDiag := P_Sample.stSafeDiag)
    Frame (300,0 1050x500)
        shows PH_SafeDiag_DiagHistory_black()
END_VISUALIZATION
